SUBAPPLICATION Uebung_024 (* Spiegelabfolge (4) *)
  (* Standard: 61499-2; Description: Copyright (c) 2023 Meisterschulen am Ostbahnhof This program and the accompanying materials are made available under the terms of the Eclipse Public License 2.0 which is available at https://www.eclipse.org/legal/epl-2.0/ SPDX-License-Identifier: EPL-2.0 *)
  (* Version 1.0, 2023-10-23, Franz Höpfinger, Meisterschulen am Ostbahnhof *)
  IMPORT SoftKeyActivationCode::SK_PRESSED;
  IMPORT SoftKeyActivationCode::SK_RELEASED;
  IMPORT Uebungen::const::UT::DefaultPool::SoftKey_F1;
  IMPORT Uebungen::const::UT::DefaultPool::SoftKey_F2;
  IMPORT Uebungen::const::UT::DefaultPool::SoftKey_F3;
  IMPORT Uebungen::const::UT::DefaultPool::SoftKey_F8;
  IMPORT Uebungen::const::UT::DefaultPool::SoftKey_F9;
  IMPORT logiBUS::io::DQ::logiBUS_DO::Output_Q1;
  IMPORT logiBUS::io::DQ::logiBUS_DO::Output_Q2;
  IMPORT logiBUS::io::DQ::logiBUS_DO::Output_Q3;
  IMPORT logiBUS::io::DQ::logiBUS_DO::Output_Q4;
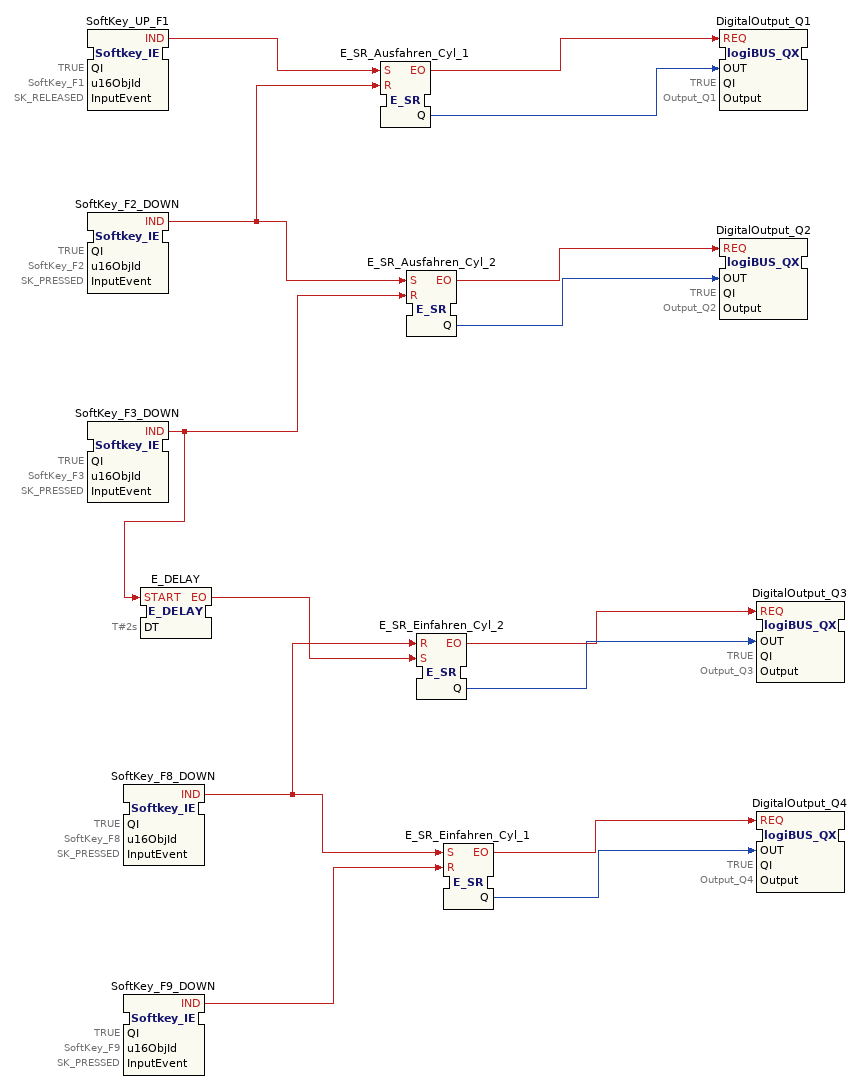
  (* START-Knopf Ausfahren *)
  (* Endlage Ausfahren_Cyl_1 *)
  (* Endlage Ausfahren_Cyl_2 *)
  (* Ausfahren_Cyl_1 *)
  (* Ausfahren_Cyl_2 *)
  (* Einfahren Zeit gesteuert *)
  (* Endlage Einfahren_Cyl_1 *)
  (* Einfahren_Cyl_2 *)
  (* Endlage Einfahren_Cyl_2 *)
  (* Einfahren_Cyl_1 *)
  FBS
    DigitalOutput_Q1 : logiBUS::io::DQ::logiBUS_QX(QI := TRUE, Output := Output_Q1);
    SoftKey_UP_F1 : Softkey_IE(QI := TRUE, u16ObjId := SoftKey_F1, InputEvent := SK_RELEASED);
    E_SR_Ausfahren_Cyl_1 : iec61499::events::E_SR;
    SoftKey_F2_DOWN : Softkey_IE(QI := TRUE, u16ObjId := SoftKey_F2, InputEvent := SK_PRESSED);
    DigitalOutput_Q2 : logiBUS::io::DQ::logiBUS_QX(QI := TRUE, Output := Output_Q2);
    E_SR_Ausfahren_Cyl_2 : iec61499::events::E_SR;
    SoftKey_F3_DOWN : Softkey_IE(QI := TRUE, u16ObjId := SoftKey_F3, InputEvent := SK_PRESSED);
    SoftKey_F9_DOWN : Softkey_IE(QI := TRUE, u16ObjId := SoftKey_F9, InputEvent := SK_PRESSED);
    E_SR_Einfahren_Cyl_2 : iec61499::events::E_SR;
    DigitalOutput_Q3 : logiBUS::io::DQ::logiBUS_QX(QI := TRUE, Output := Output_Q3);
    DigitalOutput_Q4 : logiBUS::io::DQ::logiBUS_QX(QI := TRUE, Output := Output_Q4);
    E_SR_Einfahren_Cyl_1 : iec61499::events::E_SR;
    SoftKey_F8_DOWN : Softkey_IE(QI := TRUE, u16ObjId := SoftKey_F8, InputEvent := SK_PRESSED);
    E_DELAY : iec61499::events::E_DELAY(DT := T#2s);
  END_FBS
  EVENT_CONNECTIONS
    SoftKey_UP_F1.IND TO E_SR_Ausfahren_Cyl_1.S;
    SoftKey_F2_DOWN.IND TO E_SR_Ausfahren_Cyl_1.R;
    E_SR_Ausfahren_Cyl_1.EO TO DigitalOutput_Q1.REQ;
    E_SR_Ausfahren_Cyl_2.EO TO DigitalOutput_Q2.REQ;
    SoftKey_F2_DOWN.IND TO E_SR_Ausfahren_Cyl_2.S;
    SoftKey_F3_DOWN.IND TO E_SR_Ausfahren_Cyl_2.R;
    E_SR_Einfahren_Cyl_2.EO TO DigitalOutput_Q3.REQ;
    SoftKey_F8_DOWN.IND TO E_SR_Einfahren_Cyl_1.S;
    E_SR_Einfahren_Cyl_1.EO TO DigitalOutput_Q4.REQ;
    SoftKey_F9_DOWN.IND TO E_SR_Einfahren_Cyl_1.R;
    SoftKey_F8_DOWN.IND TO E_SR_Einfahren_Cyl_2.R;
    E_DELAY.EO TO E_SR_Einfahren_Cyl_2.S;
    SoftKey_F3_DOWN.IND TO E_DELAY.START;
  END_CONNECTIONS
  DATA_CONNECTIONS
    E_SR_Ausfahren_Cyl_1.Q TO DigitalOutput_Q1.OUT;
    E_SR_Ausfahren_Cyl_2.Q TO DigitalOutput_Q2.OUT;
    E_SR_Einfahren_Cyl_1.Q TO DigitalOutput_Q4.OUT;
    E_SR_Einfahren_Cyl_2.Q TO DigitalOutput_Q3.OUT;
  END_CONNECTIONS
END_SUBAPPLICATION
